Staubli VAL3: onExit.pgx

program onExit()
  local string l_sMessage
begin
  //
end
